{attribute addProperty BoxType "KL3044-0001"}
{attribute addProperty Id "Channel_100Channel_200Channel_300Channel_400"}
{attribute addProperty CRC "1370403366"}
{attribute addProperty SizeInBites "0"}
{attribute addProperty SizeInBytes "0"}
TYPE KL_51AEB226 :
STRUCT
	{attribute addProperty Name "Channel_1"}
	Channel_1 : ;
	{attribute addProperty Name "Channel_2"}
	Channel_2 : ;
	{attribute addProperty Name "Channel_3"}
	Channel_3 : ;
	{attribute addProperty Name "Channel_4"}
	Channel_4 : ;
END_STRUCT
END_TYPE

(* stored: Version 1.2.0.0, ProductVersion 3.1.4024.9
   DUT KL_51AEB226: Id {e3cc9e2f-e3ec-437e-8163-5a3572af5fa4} *)
